PROGRAM MAIN
VAR
END_VAR

END_PROGRAM

(* stored: Version 1.1.0.1
   POU MAIN: Id {d6696e7a-bd8d-4b12-9aae-d25bd828de68} *)
